// Mitsubishi GX Works2 project: 플리커_카운터2   PLC: Q03UDV

// global labels: Global1
VAR_GLOBAL
  PB1 AT X15 : BOOL;
  PB2 AT X16 : BOOL;
  RED AT Y2B : BOOL;
END_VAR

PROGRAM MAIN
VAR
  TEMP : BOOL;
  타이머1 : TIMER;
  타이머2 : TIMER;
  카운터1 : COUNTER;
END_VAR
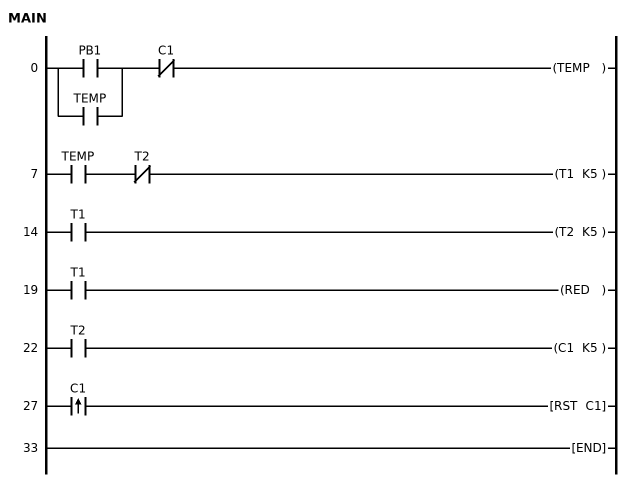
0     LD      PB1
      OR      TEMP
      ANI     C1
      OUT     TEMP
7     LD      TEMP
      ANI     T2
      OUT     T1 K5
14    LD      T1
      OUT     T2 K5
19    LD      T1
      OUT     RED
22    LD      T2
      OUT     C1 K5
27    LDP     C1
      RST     C1
33    END
END_PROGRAM
